Staubli VAL3: onF2Event.pgx

program onF2Event()
  local string l_sPath
  local string l_sItems[2]
begin
  // look if the bButton is enable
  if bButton[1]
    //
  endIf
end
